// TIA Portal V19 export
TYPE "C103_VAR_IF_OVB_TYPIC"
   STRUCT
      SCL { ExternalAccessible := 'False'; ExternalVisible := 'False'; ExternalWritable := 'False'} : Bool;   // Standmelding ingangszone 400V/230V
   END_STRUCT;
END_TYPE
